(* Logix 5000 project; controller ECE4350_Lab9_LefeversAngelino 5069-L306ERM rev 30.11; software revision 30.00 *)

TASK MainTask (continuous, watchdog 500 ms) : MainProgram

MODULES
   Local : 5069-L306ERM (5069 0, rev 30.11)
      Digital_IN : 5069-IB16 (5069 1, rev 2.1, StandardDataDriven RPI 5 ms)
      Analog_IN : vendor 1 type 115 code 314 (5069 2, rev 2.1, StandardDataDriven RPI 100 ms)
      Analog_OUT : vendor 1 type 115 code 320 (5069 4, rev 2.1, StandardDataDriven RPI 80 ms)   // Unused in this program
      Digital_OUT : 5069-OB16 (5069 3, rev 2.1, StandardDataDriven RPI 5 ms)
END_MODULES

PROGRAM MainProgram   (* main routine MainRoutine *)
VAR
   DegreesCelsius : DINT;   // Final Degrees Celsius
   GreenLED : ALIAS FOR Local:3:O.Pt00.Data;   // green led light
   int0 : DINT;   // Intermediate Variable used in Algorithm (Voltage->Celsius)
   int1 : DINT;   // Intermediate Variable used in Algorithm (Votage->Celsius)
   int2 : DINT;   // Intermediate Variable used in Algorithm (Voltage->Celsius)
   int3 : DINT;   // Intermediate Variable used in Algorithm (Voltage->Celsius)
   int4 : DINT;   // Intermediate Variable used in Algorithm (Voltage->Celsius)
   LA_Polarity : ALIAS FOR Local:3:O.Pt03.Data;   // ON: Left to Right OFF: Right to Left
   LA_POS : DINT;   // The position of the linear actuator
   LA_Power : ALIAS FOR Local:3:O.Pt05.Data;   // Linear Actuator power
   LA_Stop : BOOL;   // Allows a HMI program to stop the LA at anytime
   LA_Time : INT;   // The total amout of time it takes the LA to move from stop to stop
   LeftStop : ALIAS FOR Local:1:I.Pt04.Data;   // Left stop reed switch
   LRA : BOOL;   // Left to Right Activator Allows a HMI to move the LA from left to right
   LRF : BOOL;   // Left to Right Flag Is activated when the LA is moving from left to right
   LSO : BOOL;   // Left Stop Oneshot
   Motor : ALIAS FOR Local:3:O.Pt02.Data;
   MOTOR_OFF : BOOL;   // Gear head motor deactivation HMI Interface
   MOTOR_ON : BOOL;   // Gear head motor activate HMI Interface
   PB_Green : ALIAS FOR Local:1:I.Pt01.Data;   // Normally Off
   PB_Red : ALIAS FOR Local:1:I.Pt00.Data;   // Normally On
   POS_T : TIMER := (PRE := 1);   // Position Timer
   PositionTransducer : ALIAS FOR Local:2:I.Ch02.Data;   // Transducer which measures the angle of the gear head motor
   Potentiometer : ALIAS FOR Local:2:I.Ch00.Data;
   PSF : BOOL;   // Program Setup Initiated Flag
   PSO : BOOL;   // Program Setup Oneshot
   PST : TIMER := (PRE := 100000);   // Program Setup Timer
   PTSF : BOOL;   // Program Timing Setup Flag
   RedLED : ALIAS FOR Local:3:O.Pt01.Data;
   RightStop : ALIAS FOR Local:1:I.Pt05.Data;
   RLA : BOOL;   // Right to Left Activator Allows a HMI to move the LA from right to left
   RLF : BOOL;   // Right to Left Flag Is activated when the LA is moving from right to left
   RSO : BOOL := 1;   // Right Stop Oneshot
   ServoMotor : ALIAS FOR Local:4:O.Ch00.Data;   // Servo Motor
   SETUP_HMI : BOOL;   // Allows the HMI to enter setup mode using a LATCHED module
   Solenoid : ALIAS FOR Local:3:O.Pt06.Data;
   Temperature_HIGH : DINT;   // Reference Termperature High
   Temperature_LOW : DINT;   // Reference Temperature Low
   TemperatureAlarmFlag : BOOL;   // Stops the linear actuactor if the temperature rises above 15 degrees celsius
   Thermistor : ALIAS FOR Local:2:I.Ch01.Data;
   ThermistorVoltage_HIGH : DINT;   // Thermistor Reference Voltage - High Temperature
   ThermistorVoltage_LOW : DINT;   // Thermistor Reference Voltage - Low Temperature
   ToggleLeft : ALIAS FOR Local:1:I.Pt03.Data;   // Toggle Switch in Left Position
   ToggleRight : ALIAS FOR Local:1:I.Pt02.Data;   // Toggle Switch in Right Position
   Trans_POS : DINT;   // Holds the value from the position transducer
END_VAR

ROUTINE MainRoutine   (* ladder *)
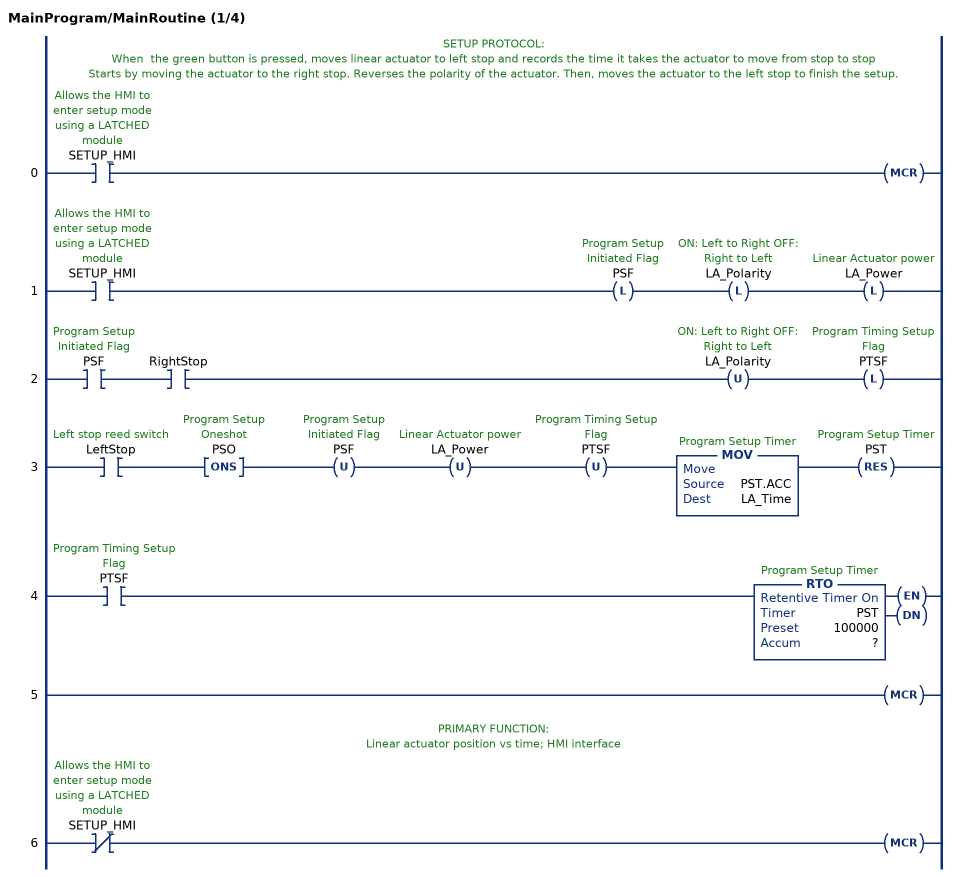
   // SETUP PROTOCOL:
   // When  the green button is pressed, moves linear actuator to left stop and records the time it takes the actuator to move from stop to stop
   // Starts by moving the actuator to the right stop. Reverses the polarity of the actuator. Then, moves the actuator to the left stop to finish the setup.
   0: XIC(SETUP_HMI)MCR();
   1: XIC(SETUP_HMI)OTL(PSF)OTL(LA_Polarity)OTL(LA_Power);
   2: XIC(PSF)XIC(RightStop)OTU(LA_Polarity)OTL(PTSF);
   3: XIC(LeftStop)ONS(PSO)OTU(PSF)OTU(LA_Power)OTU(PTSF)MOV(PST.ACC,LA_Time)RES(PST);
   4: XIC(PTSF)RTO(PST,?,?);
   5: MCR();
   // PRIMARY FUNCTION:
   // Linear actuator position vs time; HMI interface
   6: XIO(SETUP_HMI)MCR();
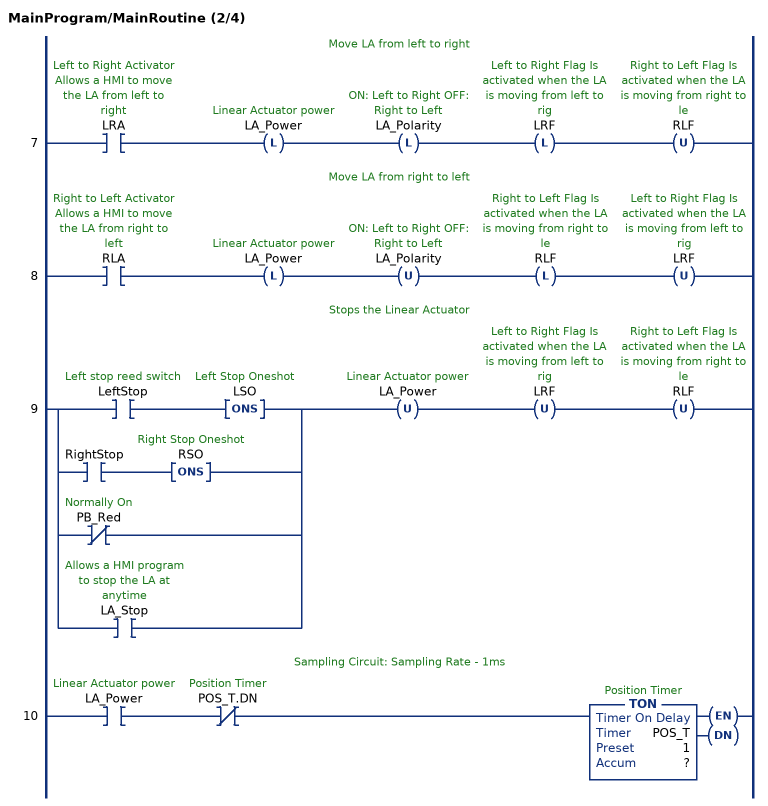
   // Move LA from left to right
   7: XIC(LRA)OTL(LA_Power)OTL(LA_Polarity)OTL(LRF)OTU(RLF);
   // Move LA from right to left
   8: XIC(RLA)OTL(LA_Power)OTU(LA_Polarity)OTL(RLF)OTU(LRF);
   // Stops the Linear Actuator
   9: [XIC(LeftStop) ONS(LSO) ,XIC(RightStop) ONS(RSO) ,XIO(PB_Red) ,XIC(LA_Stop) ]OTU(LA_Power)OTU(LRF)OTU(RLF);
   // Sampling Circuit: Sampling Rate - 1ms
   10: XIC(LA_Power)XIO(POS_T.DN)TON(POS_T,?,?);
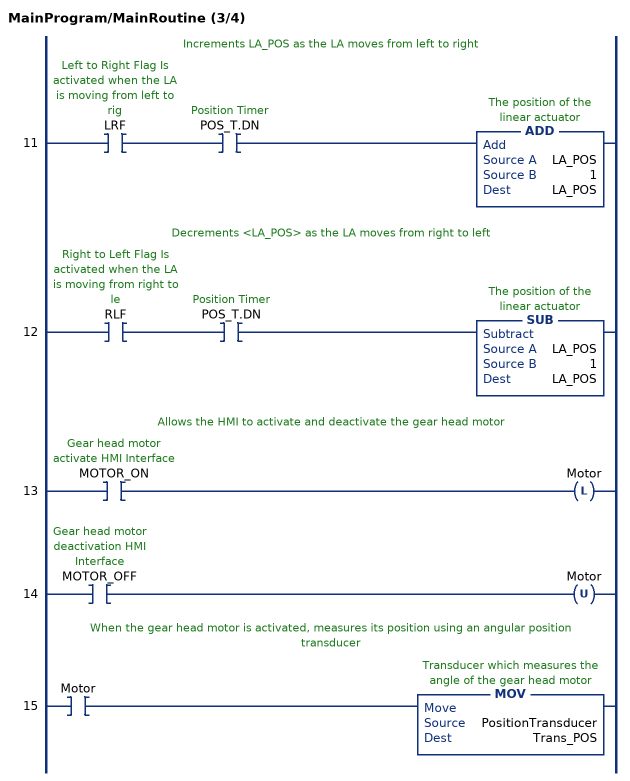
   // Increments LA_POS as the LA moves from left to right
   11: XIC(LRF)XIC(POS_T.DN)ADD(LA_POS,1,LA_POS);
   // Decrements <LA_POS> as the LA moves from right to left
   12: XIC(RLF)XIC(POS_T.DN)SUB(LA_POS,1,LA_POS);
   // Allows the HMI to activate and deactivate the gear head motor
   13: XIC(MOTOR_ON)OTL(Motor);
   14: XIC(MOTOR_OFF)OTU(Motor);
   // When the gear head motor is activated, measures its position using an angular position transducer
   15: XIC(Motor)MOV(PositionTransducer,Trans_POS);
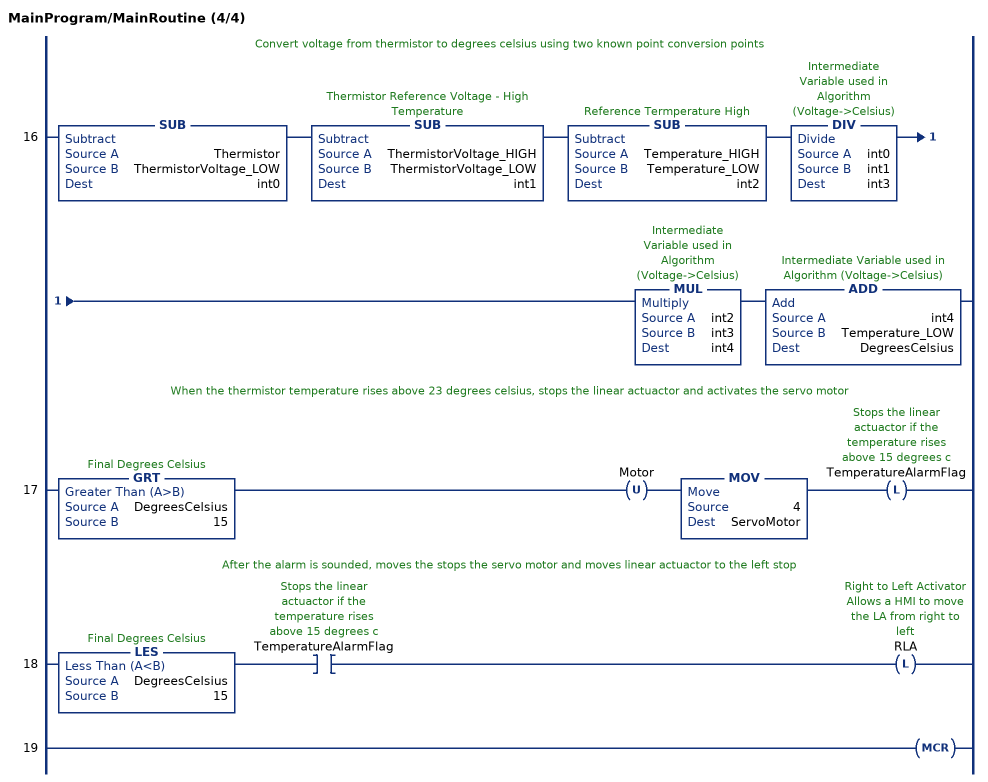
   // Convert voltage from thermistor to degrees celsius using two known point conversion points
   16: SUB(Thermistor,ThermistorVoltage_LOW,int0)SUB(ThermistorVoltage_HIGH,ThermistorVoltage_LOW,int1)SUB(Temperature_HIGH,Temperature_LOW,int2)DIV(int0,int1,int3)MUL(int2,int3,int4)ADD(int4,Temperature_LOW,DegreesCelsius);
   // When the thermistor temperature rises above 23 degrees celsius, stops the linear actuactor and activates the servo motor
   17: GRT(DegreesCelsius,15)OTU(Motor)MOV(4,ServoMotor)OTL(TemperatureAlarmFlag);
   // After the alarm is sounded, moves the stops the servo motor and moves linear actuactor to the left stop
   18: LES(DegreesCelsius,15)XIC(TemperatureAlarmFlag)OTL(RLA);
   19: MCR();
END_ROUTINE
END_PROGRAM
